Staubli VAL3: TrajHome.dtx

public num nIndexTool
public TrajJointItem tData
  [0]
    jointRx jJoint
    TrajectoryItem tSuper
      [0]
        num distance
        num moveType
        num nTime
        num nStop
        num nTcpAction
        string comment
        bool toStop
        mdesc nom_speed = {vel=50, tmax=500}
        InstrItem iInstr[3]
          [0]
            string sType
            string sData
          [1]
            string sType
            string sData
          [2]
            string sType
            string sData
        num nMoveId
public string sID
public num nZoneType
public num nZoneMove
public pointRx pO = {fatherId=world[0]}
public pointRx pX = {fatherId=world[0]}
public pointRx pY = {fatherId=world[0]}
public num nDimension
public pointRx pPointMove = {fatherId=fFrame[0]}
public frame fFrame = {fatherId=world[0]}
public string sProgram
public num nIndexFrame
